// TIA Portal V19 export
TYPE "LEXCHANGETRAY_typeTrayMonitor"
// stored: Access Published
   STRUCT
      status : "LEXCHANGETRAY_typeTrayStatus";   // 托盘状态
      postion : "LEXCHANGETRAY_typeTrayPosition";   // 托盘位置
      cellsInfo { S7_SetPoint := 'True'} : "LEXCHANGETRAY_typeCellsMonitor";
      trayCode { S7_SetPoint := 'True'} : WString;
      curScratchCellRow { S7_SetPoint := 'True'} : Int;   // 当前抓取电池的行
   END_STRUCT;
END_TYPE
